FUNCTION_BLOCK XTSHardware_V2 EXTENDS CyclicBase IMPLEMENTS I_Initialise
VAR
	XtsParts : ARRAY[0..SystemParameters.NumberOfParts-1] OF XtsPart;
	XtsTracks : ARRAY[0..SystemParameters.NumberOfTracks-1] OF XtsTrack;
	TrackOTCIDs: ARRAY [1..Tc3_XTS_Utility.TcIoXtsEnvironmentParameterList.MaxXtsTracksPerXpu] OF Tc3_XTS_Utility.OTCID;
	MyXPUInterface : Tc3_XTS_Utility.I_TcIoXtsProcessingUnit;
	MyXtsIoEnvVarRef : ITF_XTSIOEnvVarWrapper;
	XtsIoEnvInitialiseState : INT;
	i: UDINT;
	MyPartCount: UDINT;
	MyTrackCount: UDINT;
	bMoverIdDetectionActive: BOOL;
	bTriggerDetect: BOOL;
	bMoverIdDetectionError: BOOL;
	bMoverIdDetected: BOOL;
END_VAR

METHOD PUBLIC  Cycle : HRESULT
VAR_INPUT
END_VAR
FOR i := 0 TO UDINT_TO_INT(MyPartCount-1) DO
	XtsParts[i].Cycle();
END_FOR
FOR i := 0 TO UDINT_TO_INT(MyTrackCount-1) DO
	XtsTracks[i].Cycle();
END_FOR
END_METHOD

METHOD getAllMoversValid : BOOL
VAR_INPUT
END_VAR
 IF MyXPUInterface.GetAreAllPositionsValid() THEN
	 getAllMoversValid := TRUE;
	 Logger.Send(TC_EVENTS.XtsHardwareEvents.AllMoversValid,'');
 END_IF
END_METHOD

METHOD getMoversDetected : BOOL
VAR_INPUT
END_VAR
IF MyXPUInterface.GetDetectedMoverCount() = MyXPUInterface.GetExpectedMoverCount() THEN
	getMoversDetected := TRUE;
	Logger.Send(TC_EVENTS.XtsHardwareEvents.ExpectedMoversDetected,UDINT_TO_STRING(MyXPUInterface.GetExpectedMoverCount()));
ELSE
	getMoversDetected := FALSE;
	Logger.Send(TC_EVENTS.XtsHardwareEvents.ExpectedMoversNotFound,'');
END_IF
END_METHOD

METHOD GetTrackByOTCID : I_XtsTrack
VAR_INPUT
	trackOTCID : OTCID;
END_VAR
FOR i := 0 TO SystemParameters.NumberOfTracks - 1 DO
	IF trackOTCID = XtsTracks[i].MyOTCID THEN
		GetTrackByOTCID := XtsTracks[i];
	END_IF
END_FOR
END_METHOD

METHOD Initialise : HRESULT
VAR_INPUT
END_VAR

VAR
	
END_VAR
CASE XtsIoEnvInitialiseState OF
	0:
		IF MyXtsIoEnvVarRef <> 0 THEN
			IF MyXtsIoEnvVarRef.IsInitialised() THEN
				MyXPUInterface := MyXtsIoEnvVarRef.GetXPUInterface();
				XtsIoEnvInitialiseState := 1;
			END_IF
		END_IF
	1:
		MyPartCount := MyXPUInterface.GetPartCount();
		IF MyPartCount = SystemParameters.NumberOfParts THEN
			FOR i := 0 TO UDINT_TO_INT(MyPartCount - 1) DO
				XtsParts[i].MyXtsIoEnvInterface := MyXPUInterface.PartTcIo(UDINT_TO_UINT(i + 1));
				IF THIS^.IsInSim() THEN
					XtsParts[i].SetInSim();
				END_IF
			END_FOR
			XtsIoEnvInitialiseState := 3;
		ELSE
			XtsIoEnvInitialiseState := 999;
		END_IF
	3:
		MyTrackCount := MyXPUInterface.GetTrackCount();
		MyXPUInterface.GetTrackOids();
		TrackOTCIDs := MyXPUInterface.P_TrackOids;
		IF MyTrackCount = SystemParameters.NumberOfTracks THEN
			FOR i := 0 TO UDINT_TO_INT(MyTrackCount - 1) DO
				XtsTracks[i].MyXtsIoEnvInterface := MyXPUInterface.TrackTcIo(UDINT_TO_UINT(i + 1));
				XtsTracks[i].MyOTCID := TrackOTCIDs[i + 1];
			END_FOR
			XtsIoEnvInitialiseState := 4;
		ELSE
			XtsIoEnvInitialiseState := 999;
		END_IF
	4:
		XtsIoEnvInitialiseState := 5;
		FOR i := 0 TO UDINT_TO_INT(MyPartCount - 1) DO
			IF XtsParts[i].Initialise() <> 2 THEN
				XtsIoEnvInitialiseState := 4;
			END_IF
		END_FOR
	5:
		XtsIoEnvInitialiseState := 6;
		FOR i := 0 TO UDINT_TO_INT(MyTrackCount - 1) DO
			IF XtsTracks[i].Initialise() <> 2 THEN
				XtsIoEnvInitialiseState := 5;
			END_IF
		END_FOR
	6:
		Initialise := 2;
END_CASE
END_METHOD

METHOD Is24VdcOK : HRESULT
VAR_INPUT
END_VAR
Is24VdcOK := 2;
FOR i := 0 TO (MyXPUInterface.GetPartCount() -1) DO
	IF XtsParts[i].Is24VBusOK() = 1 THEN
		Is24VdcOK := 1;
	END_IF
END_FOR
END_METHOD

METHOD Is48VdcOK : HRESULT
VAR_INPUT
END_VAR
Is48VdcOK := 2;
FOR i := 0 TO (MyXPUInterface.GetPartCount() - 1) DO
	IF XtsParts[i].Is48VBusOK() = 1 THEN
		Is48VdcOK := 1;
	END_IF
END_FOR
END_METHOD

METHOD IsInSim : BOOL
VAR_INPUT
END_VAR
IF  MyXtsIoEnvVarRef.IsInSim() THEN
	IsInSim := TRUE;
	Logger.Send(TC_EVENTS.XtsHardwareEvents.XtsInSimulationMode,'');
ELSE
	IsInSim := FALSE;
END_IF
END_METHOD

PROPERTY MyXtsIoEnvVarWrapper : itf_xtsioenvvarwrapper
GET
MyXtsIoEnvVarWrapper := MyXtsIoEnvVarRef;
END_GET
SET
MyXtsIoEnvVarRef := MyXtsIoEnvVarWrapper;
END_SET
END_PROPERTY

METHOD SetTrackForDetection : BOOL
VAR_INPUT
	TrackToDetect : INT;
END_VAR
IF MyTrackCount = 1 THEN
	MyXPUInterface.TrackTcIo(1).SetIsIncludedInDetection(TRUE);
	Logger.Send(TC_EVENTS.XtsHardwareEvents.ActiveTracksAddedForDetection, UDINT_TO_STRING(MyXPUInterface.GetTrackCount()));
	SetTrackForDetection := TRUE;
ELSE
	IF TrackToDetect <= MyTrackCount THEN 
		SetTrackForDetection := TRUE;
		MyXPUInterface.TrackTcIo(TrackToDetect).SetIsIncludedInDetection(TRUE);
		Logger.Send(TC_EVENTS.XtsHardwareEvents.ActiveTracksAddedForDetection, UDINT_TO_STRING(MyXPUInterface.GetTrackCount()));
	END_IF
END_IF
END_METHOD

METHOD TriggerMoverDetection : BOOL
VAR_INPUT
END_VAR
MyXPUInterface.TriggerRedetection();
Logger.Send(TC_EVENTS.XtsHardwareEvents.MoverDetectionInitiated,'');
TriggerMoverDetection := true;
END_METHOD

METHOD TriggerMoverID : BOOL
VAR_INPUT
END_VAR
// Mover1 Functionality		
// Check if "MoverIdDetectionMode" has been activated under the XtsProcessingUnit object.
IF MyXPUInterface.GetMoverIdDetectionMode() = E_MoverIdDetectionMode.Mover1 THEN

	// Check if the "MoverIdDetection" has already been started or the Mover1 was found.
	IF NOT (bMoverIdDetectionActive OR bMoverIdDetected OR bTriggerDetect) THEN
		
		// Trigger the "MoverIdDetection".
		MyXPUInterface.TriggerMoverIdDetection();
		Logger.Send(TC_EVENTS.XtsHardwareEvents.Mover1DetectionStarted,'');
		bTriggerDetect := true;
	END_IF

	// Check for error or success of "MoverIdDetection".
	bMoverIdDetectionError 	:= MyXPUInterface.GetHasMoverIdDetectionError();
	bMoverIdDetected 	:= MyXPUInterface.GetIsMoverIdDetectionValid();
	bMoverIdDetectionActive	:= MyXPUInterface.GetIsMoverIdDetectionActive();
	
	// If the detection has an error, check for errors in output and try again.
	IF bMoverIdDetectionError THEN
		Logger.Send(TC_EVENTS.XtsHardwareEvents.Mover1DetectionFailed,'');
		RETURN; 
	END_IF

	// Do not process any further until the "MoverId" was deteced.
	IF NOT bMoverIdDetected THEN
		RETURN;
	END_IF	
	TriggerMoverID := TRUE;	
	Logger.Send(TC_EVENTS.XtsHardwareEvents.Mover1DetectionComplete,'');
ELSE
	TriggerMoverID := TRUE;
	Logger.Send(TC_EVENTS.XtsHardwareEvents.StandardMoverNumberingComplete,'');
END_IF
END_METHOD

END_FUNCTION_BLOCK

(* stored: Version 1.1.0.1
   POU XTSHardware_V2: Id {2082c175-1a19-4a3f-b920-8dbd46477756}, SpecialFunc None
   Method Cycle: Id {907368a2-7640-4dfa-a8a9-6f1d20861921}
   Method getAllMoversValid: Id {61902ec7-4049-4544-9a8e-27dabf1b61be}
   Method getMoversDetected: Id {6134912a-11cc-419f-9366-ca4c2c2c2f9f}
   Method GetTrackByOTCID: Id {d55b1037-e87a-4176-a531-719c46a289ea}
   Method Initialise: Id {95822be7-e433-46ff-bfc3-e4b3c51e2a74}
   Method Is24VdcOK: Id {16c30a69-c544-4706-ba78-c8aed5346201}
   Method Is48VdcOK: Id {ff4a117c-24f4-4466-b159-c15d29dc7330}
   Method IsInSim: Id {c26b05e6-e2eb-40cc-bea5-adcd4dafa0e7}
   Property MyXtsIoEnvVarWrapper: Id {9f0e6f27-b8f0-452c-b07d-d4d2a7ed1b3b}
   Get Get: Id {ef18a883-259a-46c5-ac1a-fd1d0138159b}
   Set Set: Id {3f18a9fd-c75b-45a9-b0a5-a4cb82b21b6b}
   Method SetTrackForDetection: Id {33a6fd5d-a8a8-4e54-be38-eeae850dd3e9}
   Method TriggerMoverDetection: Id {15e78533-ebfe-46e6-bd25-18e4044d6883}
   Method TriggerMoverID: Id {23436421-ecb3-466c-b86b-5fefe5c7904c} *)
